// TIA Portal V18 export
DATA_BLOCK "flow_measurement_ladder_DB"   // DB5
VERSION : 0.1
// stored: AutoNumber true, InstanceOfName flow_measurement, InstanceOfType FB
"flow_measurement"
   // VAR
   //    K_factor : Real;
   // END_VAR
BEGIN
END_DATA_BLOCK
